FUNCTION_BLOCK COLOR_DECIDER (* Basic Function Block Type *)
  (* Standard: 61499-2 *)
  (* Version 0.3, 2009-09-15, JHC, Holobloc Inc, Changed transition priorities. *)
  (* Version 0.2, 2003-12-04, JHC, Rockwell Automation, Renamed for better indexing. *)
  (* Version 0.1, 2002-11-05, JHC, Rockwell Automation, Corrected missing ST element in Algorithm REQ. *)
  (* Version 0.0, 2000-05-30, JHC, Rockwell Automation *)
  PACKAGE fb.rt.Conveyer;
  IMPORT fb.datatype.*;
  IMPORT fb.rt.*;
  IMPORT fb.rt.mva.VSTYLE;
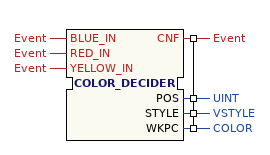
  EVENT_INPUT
    BLUE_IN;
    RED_IN;
    YELLOW_IN;
  END_EVENT
  EVENT_OUTPUT
    CNF WITH POS, STYLE, WKPC; (* Execution Confirmation *)
  END_EVENT
  VAR_OUTPUT
    POS : UINT := 0;
    STYLE : VSTYLE := PALLET;
    WKPC : COLOR;
  END_VAR
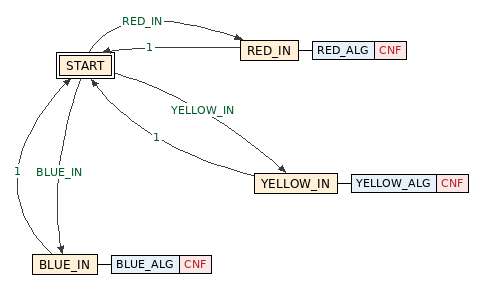
  EC_STATES
    START; (* Initial State *)
    BLUE_IN : BLUE_ALG -> CNF;
    YELLOW_IN : YELLOW_ALG -> CNF;
    RED_IN : RED_ALG -> CNF;
  END_STATES
  EC_TRANSITIONS
    START TO RED_IN := RED_IN;
    RED_IN TO START := 1;
    START TO YELLOW_IN := YELLOW_IN;
    YELLOW_IN TO START := 1;
    START TO BLUE_IN := BLUE_IN;
    BLUE_IN TO START := 1;
  END_TRANSITIONS
  ALGORITHM RED_ALG IN ST:
POS := 0;
STYLE := PALLET;
WKPC := red;
  END_ALGORITHM
  ALGORITHM BLUE_ALG IN ST:

  END_ALGORITHM
  ALGORITHM YELLOW_ALG IN ST:

  END_ALGORITHM
END_FUNCTION_BLOCK
